VAR_GLOBAL CONSTANT
    ADSLOG_MSGTYPE_HINT  : DWORD := 1;
    ADSLOG_MSGTYPE_WARN  : DWORD := 2;
    ADSLOG_MSGTYPE_ERROR : DWORD := 3;
    ADSLOG_MSGTYPE_INFO  : DWORD := 4;
END_VAR

(* stored: Version 1.1.0.1
   GVL GVL_ADSLOG: Id {9cef96f7-573a-43ca-943f-153dd8b8a3f1} *)
